(* PLC project spindle, Dassault Systèmes ControlBuild 2024x *)
(* stored: creationDateTime 2023-10-03T11:13:44-01:00 *)

FUNCTION_BLOCK drill.spindle
  VAR_INPUT
    rotation : BOOL := false;
    acknowledgePB : BOOL := false;
    equipmentFault : BOOL := false;
  END_VAR
  VAR_OUTPUT
    contactor : BOOL := false;
    rotationFault : DINT := 0;
  END_VAR

INITIAL_STEP 10:
  COMPUTE_FUNCTION_BLOCKS(S);
END_STEP
TRANSITION FROM 10 TO 11
  := rotation AND (rotationFault = 0);
END_TRANSITION
STEP 11:
  11_INLINE1(N);
END_STEP
ACTION 11_INLINE1:
  contactor;
END_ACTION
TRANSITION FROM 11 TO 10
  := NOT rotation OR (rotationFault > 0);
END_TRANSITION
ACTION COMPUTE_FUNCTION_BLOCKS:  (* blocks drawn on the SFC sheet *)
  G1:
END_ACTION

ACTION PreSFC:
IF((RE acknowledgePB)) THEN
	rotationFault := 0;
END_IF;
IF (X11 AND equipmentFault) THEN
	rotationFault := 1;
END_IF;
END_ACTION
END_FUNCTION_BLOCK
